FUNCTION_BLOCK Current_Transformer (* Composite Function Block Type *)
  (* Standard: 61499-2 *)
  (* Version 0.0, 12/10/2023, Cheyan, Schneider Electric, template *)
  PACKAGE Main;
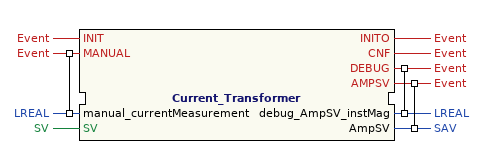
  EVENT_INPUT
    INIT; (* Initialization Request *)
    MANUAL WITH manual_currentMeasurement;
  END_EVENT
  EVENT_OUTPUT
    INITO; (* Initialization Confirm *)
    CNF; (* Execution Confirmation *)
    DEBUG WITH debug_AmpSV_instMag;
    AMPSV WITH AmpSV;
  END_EVENT
  VAR_INPUT
    manual_currentMeasurement : LREAL;
  END_VAR
  VAR_OUTPUT
    debug_AmpSV_instMag : LREAL;
    AmpSV : SAV; (* Output event qualifier *)
  END_VAR
  SOCKETS
    SV : SV;
  END_SOCKETS
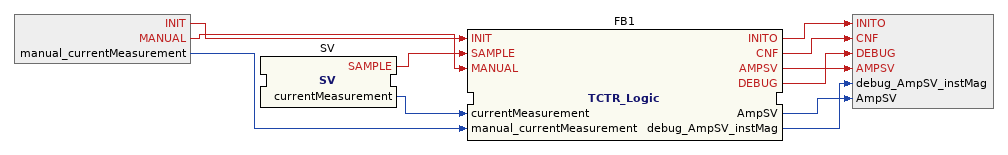
  FBS
    FB1 : TCTR_Logic;
  END_FBS
  EVENT_CONNECTIONS
    INIT TO FB1.INIT;
    FB1.INITO TO INITO;
    FB1.CNF TO CNF;
    SV.SAMPLE TO FB1.SAMPLE;
    FB1.DEBUG TO DEBUG;
    MANUAL TO FB1.MANUAL;
    FB1.AMPSV TO AMPSV;
  END_CONNECTIONS
  DATA_CONNECTIONS
    SV.currentMeasurement TO FB1.currentMeasurement;
    FB1.debug_AmpSV_instMag TO debug_AmpSV_instMag;
    manual_currentMeasurement TO FB1.manual_currentMeasurement;
    FB1.AmpSV TO AmpSV;
  END_CONNECTIONS
END_FUNCTION_BLOCK
